(* PLC project Generated.project, CODESYS CODESYS V3.5 SP19 Patch 1 *)
(* stored: creationDateTime 2026-07-29T11:10:15.670501, modificationDateTime 2026-07-29T11:10:15.670501 *)

TYPE ST_Chain_Translation_Control : STRUCT
  Idx401_MotionAllowed : BOOL;  (* 1 = Mouvement Translation Autorisé | 0 = Bloqué *)
  Idx402_SetpointFreq_Hz : REAL;  (* [Hz] Consigne Fréquence Calculée *)
  Idx403_DriveControlWord : WORD;  (* Mot de Commande Calculé Variateur AC600 *)
  Idx404_FinalInterlockState : E_State;  (* 🛡️ État frontière _LD *)
  Idx405_FinalInterlockReason : E_TranslationFinalInterlockReason;  (* 🛡️ Cause mémorisée *)
  Idx406_BrakeCommandOpenConfirmed : BOOL;  (* 🔌 Contacteur/bobine, pas frein mécanique *)
  Idx407_BrakeTimeoutElapsed : TIME;  (* ⏱️ Watchdog 500ms écoulé *)
END_STRUCT;
END_TYPE

(* values of E_State: DISABLED: Enable faux, neutralisé; INIT: Démarrage / vérifs; READY: Prêt, attend ordre; BUSY: Action en cours; DONE: Action terminée; STOPPING: Décél rampe avant arrêt (StartStop=FALSE ou SafeStop=TRUE) *)

{attribute 'qualified_only'}
{attribute 'strict'}
TYPE E_State : (DISABLED := 0, INIT := 1, READY := 2, BUSY := 3, DONE := 4, STOPPING := 5);
END_TYPE

{attribute 'qualified_only'}
{attribute 'strict'}
TYPE E_TranslationFinalInterlockReason : (NONE := 0, BRAKE_COMMAND_NOT_CONFIRMED := 1, RESTART_INHIBITED := 2);
END_TYPE
